PROGRAM T00_FAST
VAR
	bExecuteDiagnosticBlock	: BOOL;
END_VAR

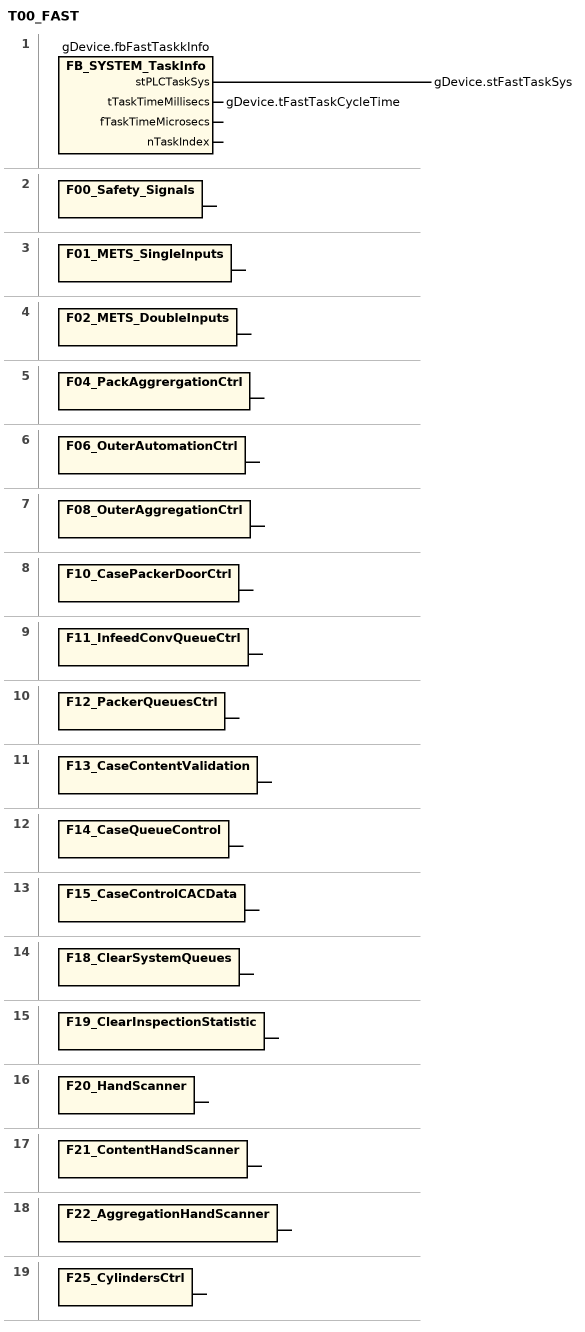
// NETWORK 1
gDevice.fbFastTaskkInfo(tTaskTimeMillisecs => gDevice.tFastTaskCycleTime); // FB_SYSTEM_TaskInfo
gDevice.stFastTaskSys := gDevice.fbFastTaskkInfo.stPLCTaskSys;

// NETWORK 2
F00_Safety_Signals();

// NETWORK 3
F01_METS_SingleInputs();

// NETWORK 4
F02_METS_DoubleInputs();

// NETWORK 5
F04_PackAggrergationCtrl();

// NETWORK 6
F06_OuterAutomationCtrl();

// NETWORK 7
F08_OuterAggregationCtrl();

// NETWORK 8
F10_CasePackerDoorCtrl();

// NETWORK 9
F11_InfeedConvQueueCtrl();

// NETWORK 10
F12_PackerQueuesCtrl();

// NETWORK 11
F13_CaseContentValidation();

// NETWORK 12
F14_CaseQueueControl();

// NETWORK 13
F15_CaseControlCACData();

// NETWORK 14
F18_ClearSystemQueues();

// NETWORK 15
F19_ClearInspectionStatistic();

// NETWORK 16
F20_HandScanner();

// NETWORK 17
F21_ContentHandScanner();

// NETWORK 18
F22_AggregationHandScanner();

// NETWORK 19
F25_CylindersCtrl();

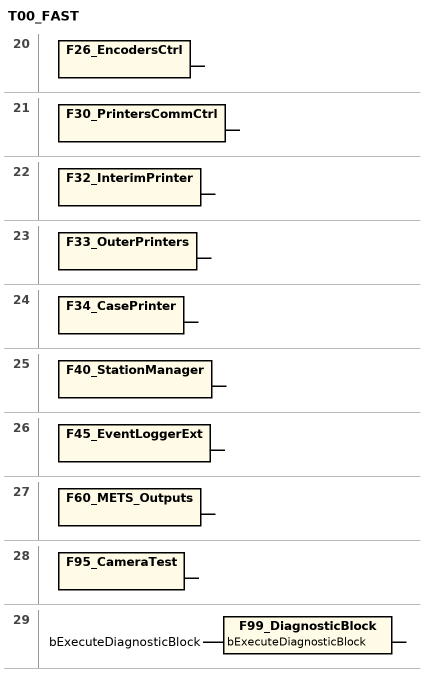
// NETWORK 20
F26_EncodersCtrl();

// NETWORK 21
F30_PrintersCommCtrl();

// NETWORK 22
F32_InterimPrinter();

// NETWORK 23
F33_OuterPrinters();

// NETWORK 24
F34_CasePrinter();

// NETWORK 25
F40_StationManager();

// NETWORK 26
F45_EventLoggerExt();

// NETWORK 27
F60_METS_Outputs();

// NETWORK 28
F95_CameraTest();

// NETWORK 29
F99_DiagnosticBlock(bExecuteDiagnosticBlock := bExecuteDiagnosticBlock);

END_PROGRAM

(* stored: Version 1.1.0.1
   POU T00_FAST: Id {5c3e3e05-81b8-4935-a7fc-c993192f70f5}, SpecialFunc None *)
